TYPE "SetPoint"
VERSION : 0.1
   STRUCT
      Lower : "Val";
      Upper : "Val";
   END_STRUCT;

END_TYPE

